PROGRAM PRG_Test
VAR
	comparisonFunctionsTest : ComparisonFunctionsTest;
	compareAnyTypeTest : CompareAnyTypeTest;
	
	manipulateFunctionsTest : ManipulateFunctionsTest;
	quickSortFunctionsTest : QuickSortFunctionsTest;
	SortFunctionsTest : SortFunctionsTest;

	tableSerializerTest : TableSerializerTest;
	tableDeserializerTest : TableDeserializerTest;
END_VAR

TcUnit.RUN();

END_PROGRAM

(* stored: Version 1.1.0.1, ProductVersion 3.1.4024.15
   POU PRG_Test: Id {380864e4-85d3-01fc-242a-a3eab7227cbd}, SpecialFunc None *)
